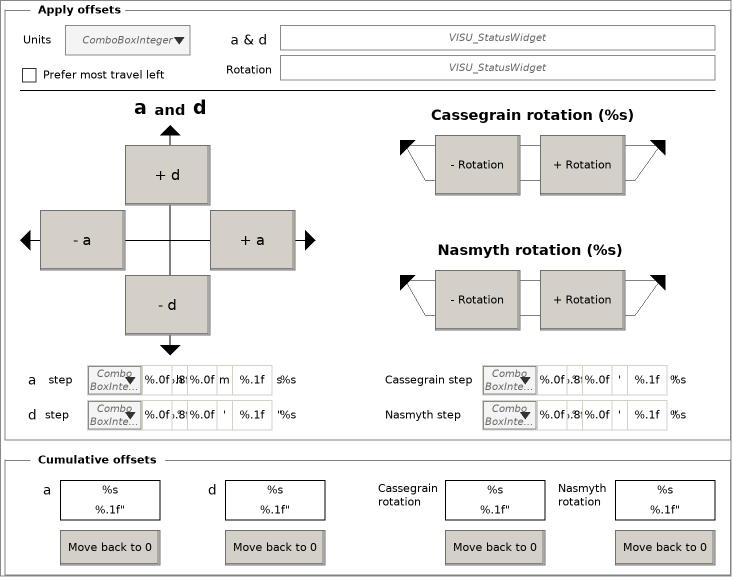
VISUALIZATION VISU_AxesManual_Offsets_AlphaDeltaRot  // 732x577
VAR_IN_OUT
	ref : Axes;
    widget : AxesManualOffsetsWidget;
END_VAR
    Polyline (165,460) (730,460) (730,575) (5,575) (5,460) (30,460)
    Polyline (125,10) (730,10) (730,440) (5,440) (5,10) (30,10)
    Polygon (660,145) (635,180) (425,180) (405,145)
    Line (170,350) (170,130)
    Line (25,240) (315,240)
    ComboBoxInteger (65,25 125x30), variable: widget.moveRelative.units, text list: 'AxesMoveAlphaDeltaProcessUnitsTextList'
    Rectangle (277,365 35x30), "%s", text variable: widget.pointRelative.unitsText, invisible if: widget.pointRelative.units = AxesMoveProcessWidgetUnits.DEGMINSEC
    Textfield (87,365 180x30), "%.8f", text variable: widget.pointRelative.field_alpha_decimal, invisible if: widget.pointRelative.units = AxesMoveProcessWidgetUnits.DEGMINSEC, input disabled if: widget.pointRelative.alphaDisabled
        OnMouseClick: write the text variable via VisuDialogs.Numpad
    Textfield (142,365 30x30), "%.0f", text variable: widget.pointRelative.field_alpha_h, invisible if: widget.pointRelative.units <> AxesMoveProcessWidgetUnits.DEGMINSEC, input disabled if: widget.pointRelative.alphaDisabled
        OnMouseClick: write the text variable via VisuDialogs.Numpad
    ComboBoxInteger (88,366 53x28), variable: widget.pointRelative.field_alpha_sign, invisible if: widget.pointRelative.units <> AxesMoveProcessWidgetUnits.DEGMINSEC, input disabled if: widget.pointRelative.alphaDisabled, text list: 'AxesDialogSignTextList'
    Textfield (187,365 30x30), "%.0f", text variable: widget.pointRelative.field_alpha_m, invisible if: widget.pointRelative.units <> AxesMoveProcessWidgetUnits.DEGMINSEC, input disabled if: widget.pointRelative.alphaDisabled
        OnMouseClick: write the text variable via VisuDialogs.Numpad
    Textfield (232,365 40x30), "%.1f", text variable: widget.pointRelative.field_alpha_s, invisible if: widget.pointRelative.units <> AxesMoveProcessWidgetUnits.DEGMINSEC, input disabled if: widget.pointRelative.alphaDisabled
        OnMouseClick: write the text variable via VisuDialogs.Numpad
    Label (172,365 15x30), "h", invisible if: widget.moveRelative.units <> AxesMoveProcessWidgetUnits.DEGMINSEC
    Label (217,365 15x30), "m", invisible if: widget.pointRelative.units <> AxesMoveProcessWidgetUnits.DEGMINSEC
    Label (272,365 15x30), "s", invisible if: widget.pointRelative.units <> AxesMoveProcessWidgetUnits.DEGMINSEC
    Rectangle (277,400 35x30), "%s", text variable: widget.pointRelative.unitsText, invisible if: widget.pointRelative.units = AxesMoveProcessWidgetUnits.DEGMINSEC
    Textfield (87,400 180x30), "%.8f", text variable: widget.pointRelative.field_delta_decimal, invisible if: widget.pointRelative.units = AxesMoveProcessWidgetUnits.DEGMINSEC, input disabled if: widget.pointRelative.deltaDisabled
        OnMouseClick: write the text variable via VisuDialogs.Numpad
    Textfield (142,400 30x30), "%.0f", text variable: widget.pointRelative.field_delta_d, invisible if: widget.pointRelative.units <> AxesMoveProcessWidgetUnits.DEGMINSEC, input disabled if: widget.pointRelative.deltaDisabled
        OnMouseClick: write the text variable via VisuDialogs.Numpad
    ComboBoxInteger (88,401 53x28), variable: widget.pointRelative.field_delta_sign, invisible if: widget.pointRelative.units <> AxesMoveProcessWidgetUnits.DEGMINSEC, input disabled if: widget.pointRelative.deltaDisabled, text list: 'AxesDialogSignTextList'
    Textfield (187,400 30x30), "%.0f", text variable: widget.pointRelative.field_delta_m, invisible if: widget.pointRelative.units <> AxesMoveProcessWidgetUnits.DEGMINSEC, input disabled if: widget.pointRelative.deltaDisabled
        OnMouseClick: write the text variable via VisuDialogs.Numpad
    Textfield (232,400 40x30), "%.1f", text variable: widget.pointRelative.field_delta_s, invisible if: widget.pointRelative.units <> AxesMoveProcessWidgetUnits.DEGMINSEC, input disabled if: widget.pointRelative.deltaDisabled
        OnMouseClick: write the text variable via VisuDialogs.Numpad
    Label (172,400 15x30), "°", invisible if: widget.moveRelative.units <> AxesMoveProcessWidgetUnits.DEGMINSEC
    Label (217,400 15x30), "'", invisible if: widget.moveRelative.units <> AxesMoveProcessWidgetUnits.DEGMINSEC
    Label (272,400 15x30), """, invisible if: widget.pointRelative.units <> AxesMoveProcessWidgetUnits.DEGMINSEC
    Rectangle (667,365 35x30), "%s", text variable: widget.moveRelative.unitsText, invisible if: widget.moveRelative.units = AxesMoveProcessWidgetUnits.DEGMINSEC
    Textfield (482,365 180x30), "%.8f", text variable: widget.moveRelative.field_roc_decimal, invisible if: widget.moveRelative.units = AxesMoveProcessWidgetUnits.DEGMINSEC, input disabled if: widget.moveRelative.rocDisabled
        OnMouseClick: write the text variable via VisuDialogs.Numpad
    Textfield (537,365 30x30), "%.0f", text variable: widget.moveRelative.field_roc_d, invisible if: widget.moveRelative.units <> AxesMoveProcessWidgetUnits.DEGMINSEC, input disabled if: widget.moveRelative.rocDisabled
        OnMouseClick: write the text variable via VisuDialogs.Numpad
    ComboBoxInteger (483,366 53x28), variable: widget.moveRelative.field_roc_sign, invisible if: widget.moveRelative.units <> AxesMoveProcessWidgetUnits.DEGMINSEC, input disabled if: widget.moveRelative.rocDisabled, text list: 'AxesDialogSignTextList'
    Textfield (582,365 30x30), "%.0f", text variable: widget.moveRelative.field_roc_m, invisible if: widget.moveRelative.units <> AxesMoveProcessWidgetUnits.DEGMINSEC, input disabled if: widget.moveRelative.rocDisabled
        OnMouseClick: write the text variable via VisuDialogs.Numpad
    Textfield (627,365 40x30), "%.1f", text variable: widget.moveRelative.field_roc_s, invisible if: widget.moveRelative.units <> AxesMoveProcessWidgetUnits.DEGMINSEC, input disabled if: widget.moveRelative.rocDisabled
        OnMouseClick: write the text variable via VisuDialogs.Numpad
    Label (567,365 15x30), "°", invisible if: widget.moveRelative.units <> AxesMoveProcessWidgetUnits.DEGMINSEC
    Label (612,365 15x30), "'", invisible if: widget.moveRelative.units <> AxesMoveProcessWidgetUnits.DEGMINSEC
    Label (667,365 15x30), """, invisible if: widget.moveRelative.units <> AxesMoveProcessWidgetUnits.DEGMINSEC
    Rectangle (667,400 35x30), "%s", text variable: widget.moveRelative.unitsText, invisible if: widget.moveRelative.units = AxesMoveProcessWidgetUnits.DEGMINSEC
    Textfield (482,400 180x30), "%.8f", text variable: widget.moveRelative.field_ron_decimal, invisible if: widget.moveRelative.units = AxesMoveProcessWidgetUnits.DEGMINSEC, input disabled if: widget.moveRelative.ronDisabled
        OnMouseClick: write the text variable via VisuDialogs.Numpad
    Textfield (537,400 30x30), "%.0f", text variable: widget.moveRelative.field_ron_d, invisible if: widget.moveRelative.units <> AxesMoveProcessWidgetUnits.DEGMINSEC, input disabled if: widget.moveRelative.ronDisabled
        OnMouseClick: write the text variable via VisuDialogs.Numpad
    ComboBoxInteger (483,401 53x28), variable: widget.moveRelative.field_ron_sign, invisible if: widget.moveRelative.units <> AxesMoveProcessWidgetUnits.DEGMINSEC, input disabled if: widget.moveRelative.ronDisabled, text list: 'AxesDialogSignTextList'
    Textfield (582,400 30x30), "%.0f", text variable: widget.moveRelative.field_ron_m, invisible if: widget.moveRelative.units <> AxesMoveProcessWidgetUnits.DEGMINSEC, input disabled if: widget.moveRelative.ronDisabled
        OnMouseClick: write the text variable via VisuDialogs.Numpad
    Textfield (627,400 40x30), "%.1f", text variable: widget.moveRelative.field_ron_s, invisible if: widget.moveRelative.units <> AxesMoveProcessWidgetUnits.DEGMINSEC, input disabled if: widget.moveRelative.ronDisabled
        OnMouseClick: write the text variable via VisuDialogs.Numpad
    Label (567,400 15x30), "°", invisible if: widget.moveRelative.units <> AxesMoveProcessWidgetUnits.DEGMINSEC
    Label (612,400 15x30), "'", invisible if: widget.moveRelative.units <> AxesMoveProcessWidgetUnits.DEGMINSEC
    Label (667,400 15x30), """, invisible if: widget.moveRelative.units <> AxesMoveProcessWidgetUnits.DEGMINSEC
    Frame (280,25 435x25)
        shows VISU_StatusWidget(widget := widget.pointRelative.actualStatus)
    Label (35,0 100x20), "Apply offsets"
    Button (125,145 85x60), "+ d", input disabled if: widget.pointRelative.deltaDisabled
        OnMouseClick: execute {
            ref.processes.pointRelative.request(
                alphaUnits := AxesAlphaUnits.DEGREES,
                alpha := 0.0,
                deltaunits := AxesDeltaUnits.DEGREES,
                delta := widget.pointRelative.deltaDeg);
        }
    Button (125,275 85x60), "- d", input disabled if: widget.pointRelative.deltaDisabled
        OnMouseClick: execute {
            ref.processes.pointRelative.request(
                alphaUnits := AxesAlphaUnits.DEGREES,
                alpha := 0.0,
                deltaunits := AxesDeltaUnits.DEGREES,
                delta := -widget.pointRelative.deltaDeg);
        }
    Button (210,210 85x60), "+ a", input disabled if: widget.pointRelative.alphaDisabled
        OnMouseClick: execute {
            ref.processes.pointRelative.request(
                alphaUnits := AxesAlphaUnits.DEGREES,
                alpha := widget.pointRelative.alphaDeg,
                deltaunits := AxesDeltaUnits.DEGREES,
                delta := 0.0);
        }
    Button (40,210 85x60), "- a", input disabled if: widget.pointRelative.alphaDisabled
        OnMouseClick: execute {
            ref.processes.pointRelative.request(
                alphaUnits := AxesAlphaUnits.DEGREES,
                alpha := -widget.pointRelative.alphaDeg,
                deltaunits := AxesDeltaUnits.DEGREES,
                delta := 0.0);
        }
    Label (42,365 35x30), "step"
    Label (42,400 40x30), "step"
    Button (540,135 85x60), "+ Rotation", input disabled if: widget.moveRelative.rocDisabled
        OnMouseClick: execute {
            ref.processes.moveRelative.request(
                units := AxesMoveUnits.DEGREES,
                azi := 0.0,
                ele := 0.0,
                rot := 0.0,
                roc := widget.moveRelative.rocDeg,
                ron := 0.0,
                doAzi := FALSE,
                doEle := FALSE,
                doRot := FALSE,
                doRoc := TRUE,
                doRon := FALSE,
                preferMostTravel := widget.preferMostTravel);
        }
    Button (435,135 85x60), "- Rotation", input disabled if: widget.moveRelative.rocDisabled
        OnMouseClick: execute {
            ref.processes.moveRelative.request(
                units := AxesMoveUnits.DEGREES,
                azi := 0.0,
                ele := 0.0,
                rot := 0.0,
                roc := -widget.moveRelative.rocDeg,
                ron := 0.0,
                doAzi := FALSE,
                doEle := FALSE,
                doRot := FALSE,
                doRoc := TRUE,
                doRon := FALSE,
                preferMostTravel := widget.preferMostTravel);
        }
    Polygon (160,135) (170,125) (180,135)
    Polygon (30,250) (20,240) (30,230)
    Polygon (305,250) (315,240) (305,230)
    Polygon (160,345) (170,355) (180,345)
    Polygon (665,155) (665,140) (650,140)
    Polygon (400,155) (415,140) (400,140)
    Label (382,365 100x30), "Cassegrain step"
    Label (382,400 100x30), "Nasmyth step"
    Label (20,25 55x30), "Units"
    Label (220,25 50x30), "a & d"
    Line (20,90) (715,90)
    Polygon (660,280) (635,315) (425,315) (405,280)
    Button (540,270 85x60), "+ Rotation", input disabled if: widget.moveRelative.ronDisabled
        OnMouseClick: execute {
            ref.processes.moveRelative.request(
                units := AxesMoveUnits.DEGREES,
                azi := 0.0,
                ele := 0.0,
                rot := 0.0,
                roc := 0.0,
                ron := widget.moveRelative.ronDeg,
                doAzi := FALSE,
                doEle := FALSE,
                doRot := FALSE,
                doRoc := FALSE,
                doRon := TRUE,
                preferMostTravel := widget.preferMostTravel);
        }
    Button (435,270 85x60), "- Rotation", input disabled if: widget.moveRelative.ronDisabled
        OnMouseClick: execute {
            ref.processes.moveRelative.request(
                units := AxesMoveUnits.DEGREES,
                azi := 0.0,
                ele := 0.0,
                rot := 0.0,
                roc := 0.0,
                ron := -widget.moveRelative.ronDeg,
                doAzi := FALSE,
                doEle := FALSE,
                doRot := FALSE,
                doRoc := FALSE,
                doRon := TRUE,
                preferMostTravel := widget.preferMostTravel);
        }
    Polygon (665,290) (665,275) (650,275)
    Polygon (400,290) (415,275) (400,275)
    Label (145,95 50x30), "and"
    Label (25,400 20x30), "d"
    Label (25,365 20x30), "a"
    Label (190,90 40x35), "d"
    Label (110,90 40x35), "a"
    Label (205,55 70x30), "Rotation"
    Frame (280,55 435x25)
        shows VISU_StatusWidget(widget := widget.moveRelative.actualStatus)
    Rectangle (60,480 100x20), "%s", text variable: widget.alphaOffsetted.hmsString
    Label (40,475 20x30), "a"
    Rectangle (60,500 100x20), "%.1f"", text variable: ref.target.alphaOffsetted.arcseconds.value
    Label (205,475 20x30), "d"
    Button (60,530 100x35), "Move back to 0", input disabled if: widget.pointRelative.alphaDisabled
        OnMouseClick: execute {
            ref.processes.pointRelative.request(
                alphaUnits := AxesAlphaUnits.DEGREES,
                alpha := -ref.target.alphaOffsetted.degrees.value,
                deltaunits := AxesDeltaUnits.DEGREES,
                delta := 0.0);
        }
    Label (35,450 120x20), "Cumulative offsets"
    Rectangle (60,480 100x40), colour toggle: widget.pointRelative.alphaDisabled
    Rectangle (225,480 100x20), "%s", text variable: widget.deltaOffsetted.dmsString
    Rectangle (225,500 100x20), "%.1f"", text variable: ref.target.deltaOffsetted.arcseconds.value
    Button (225,530 100x35), "Move back to 0", input disabled if: widget.pointRelative.deltaDisabled
        OnMouseClick: execute {
            ref.processes.pointRelative.request(
                alphaUnits := AxesAlphaUnits.DEGREES,
                alpha := 0.0,
                deltaunits := AxesDeltaUnits.DEGREES,
                delta := -ref.target.deltaOffsetted.degrees.value);
        }
    Rectangle (225,480 100x40), colour toggle: widget.pointRelative.deltaDisabled
    Rectangle (445,480 100x20), "%s", text variable: widget.rocTargetOffset.dmsString
    Rectangle (445,500 100x20), "%.1f"", text variable: ref.parts.roc.targetOffset.arcseconds.value
    Button (445,530 100x35), "Move back to 0", input disabled if: widget.moveRelative.rocDisabled
        OnMouseClick: execute {
            ref.processes.moveRelative.request(
                units := AxesMoveUnits.DEGREES,
                azi := 0.0,
                ele := 0.0,
                rot := 0.0,
                roc := -ref.parts.roc.targetOffset.degrees.value,
                ron := 0.0,
                doAzi := FALSE,
                doEle := FALSE,
                doRot := FALSE,
                doRoc := TRUE,
                doRon := FALSE, preferMostTravel := widget.preferMostTravel);
        }
    Rectangle (445,480 100x40), colour toggle: widget.moveRelative.rocDisabled
    Label (375,480 70x30), "Cassegrain rotation"
    Rectangle (615,480 100x20), "%s", text variable: widget.ronTargetOffset.dmsString
    Rectangle (615,500 100x20), "%.1f"", text variable: ref.parts.ron.targetOffset.arcseconds.value
    Button (615,530 100x35), "Move back to 0", input disabled if: widget.moveRelative.ronDisabled
        OnMouseClick: execute {
            ref.processes.moveRelative.request(
                units := AxesMoveUnits.DEGREES,
                azi := 0.0,
                ele := 0.0,
                rot := 0.0,
                roc := 0.0,
                ron :=  -ref.parts.ron.targetOffset.degrees.value,
                doAzi := FALSE,
                doEle := FALSE,
                doRot := FALSE,
                doRoc := FALSE,
                doRon := TRUE, preferMostTravel := widget.preferMostTravel);
        }
    Rectangle (615,480 100x40), colour toggle: widget.moveRelative.ronDisabled
    Label (555,480 60x30), "Nasmyth rotation"
    Rectangle (380,235 300x30), "Nasmyth rotation (%s)", text variable: ref.config.nasmythRotatorName
    Rectangle (380,100 305x30), "Cassegrain rotation (%s)", text variable: ref.config.cassegrainRotatorName
    Checkbox (20,60 195x30), "Prefer most travel left", variable: widget.preferMostTravel
END_VISUALIZATION

(* stored: Version 1.1.0.1, ProductVersion 3.1.4019.2
   Visu VISU_AxesManual_Offsets_AlphaDeltaRot: Id {e0bafc6e-eafd-4282-ab6b-9c792e3cfaa6} *)
